FUNCTION_BLOCK LinearSpline EXTENDS Spline
VAR_INPUT
	x: ARRAY [0..1] OF LREAL;
	y: ARRAY [0..1] OF LREAL;
END_VAR
VAR_OUTPUT
END_VAR
VAR
	init : BOOL := FALSE;
END_VAR

startPoint.x 	:= x[0];
startPoint.y 	:= y[0];

endPoint.x		:= x[1];
endPoint.y     	:= y[1];

startPoint.theta	:= ATAN2(endPoint.y-startPoint.y, endPoint.x-startPoint.x); 
lengthVar := calculateLength();

METHOD PROTECTED  calculateLength : LREAL
VAR_INPUT
END_VAR
calculateLength := SQRT(EXPT(startPoint.x - endPoint.x,2) + EXPT(startPoint.y - endPoint.y, 2))
END_METHOD

METHOD  diff : RobotPoseSimple
VAR_INPUT
	arcLength: LREAL;
	order: INT := 1;
END_VAR
IF order = 1 THEN
	RobotPoseSimple.x 		:= COS(startPoint.theta);
	RobotPoseSimple.y 		:= SIN(startPoint.theta);
	RobotPoseSimple.theta   := -1; //not used
ELSIF order = 2 THEN
	RobotPoseSimple.x 		:= 0;
	RobotPoseSimple.y 		:= 0;
	RobotPoseSimple.theta   := -1; //not used
ELSE
	//invalid input
	RobotPoseSimple.x 		:= -1; 
	RobotPoseSimple.y 		:= -1;
	RobotPoseSimple.theta   := -1; //not used
END_IF
END_METHOD

METHOD PUBLIC  getPoint : RobotPoseSimple
VAR_INPUT
	arcLength: LREAL;
END_VAR
getPoint.x		:= COS(startPoint.theta)*arcLength;
getPoint.y		:= SIN(startPoint.theta)*arcLength;
getPoint.theta  := -1; //not used
END_METHOD

END_FUNCTION_BLOCK

(* stored: Version 1.1.0.1, ProductVersion 3.1.4024.11
   POU LinearSpline: Id {ee8a5752-8731-4d20-b9ec-42a2604040d7}, SpecialFunc None
   Method calculateLength: Id {b557106d-f894-499c-b93e-4ca33bd951b4}
   Method diff: Id {b27160dd-5577-4e29-b3d1-95343ea264e1}
   Method getPoint: Id {2d494b1b-e161-44ef-b005-acd30148114d} *)
